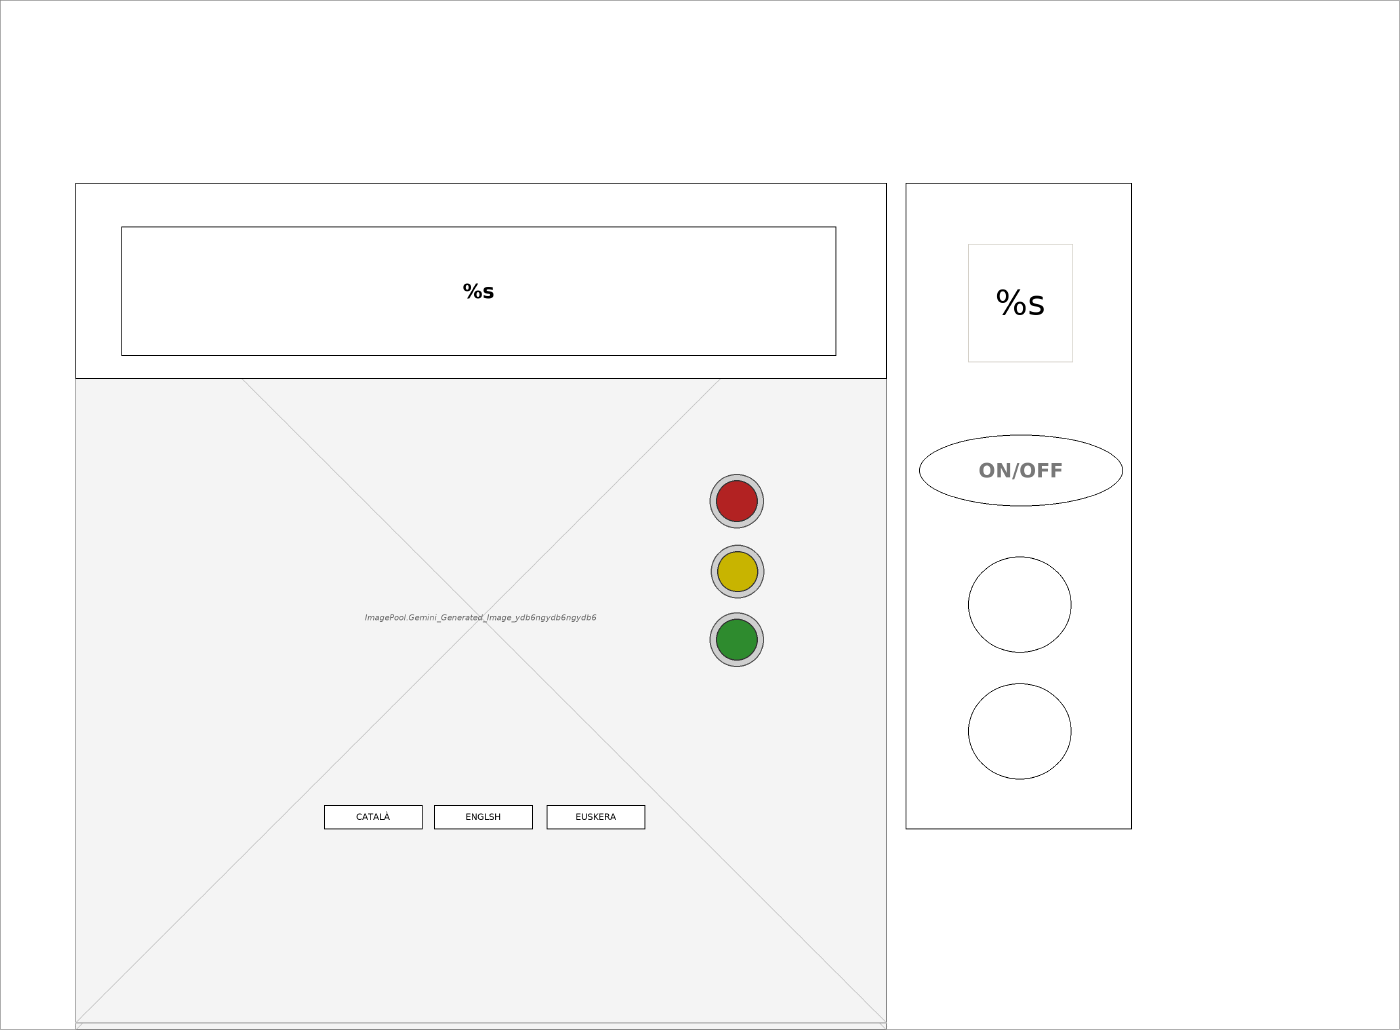
VISUALIZATION mainPage  // 1767x1301
    Image (95,272 1024x1024), invisible if: MAIN.boolENG, image: ImagePool.1772114357870
    RoundedRectangle (951,388 816x285), angle 90
    Image (95,253 1024x1048), invisible if: MAIN.boolCAT, image: ImagePool.Gemini_Generated_Image_6byr8p6byr8p6byr - copia
    Image (95,268 1024x1024), invisible if: MAIN.boolEUS, image: ImagePool.Gemini_Generated_Image_ydb6ngydb6ngydb6
    RoundedRectangle (95,231 1024x247)
    Lamp1 (890,593 80x80), variable: MAIN.mytrafficlight.outputs.REDlight, style: Lamp-Lamp1-Red
    Lamp1 (891,683 80x78), variable: MAIN.mytrafficlight.outputs.YELLOWlight, style: Lamp-Lamp1-Yellow
    Lamp1 (890,768 80x80), variable: MAIN.mytrafficlight.outputs.GREENlight, style: Lamp-Lamp1-Green
    Label (424,246 395x30), "EL HMI DEL SEMÁFORO"
    Ellipse (1222,703 130x121), colour toggle: MAIN.mytrafficlight.inputs.iGreen
        tap MAIN.mytrafficlight.inputs.iGreen
    Ellipse (1222,863 130x121), colour toggle: MAIN.mytrafficlight.inputs.iRed
        tap MAIN.mytrafficlight.inputs.iRed p1329445385=TRUE
    Ellipse (1160,549 257x90), "ON/OFF"
        toggle MAIN.updateState.HMI_Switch
    RoundedRectangle (409,1017 124x30), "CATALÀ"
        toggle MAIN.boolCAT
        OnMouseClick: ChangeLanguage ChangeLanguage=CATALÀ
        OnMouseClick: execute {
            MAIN.boolCAT := FALSE;
            MAIN.boolENG := TRUE;
            MAIN.boolEUS := TRUE;
        }
    RoundedRectangle (548,1017 124x30), "ENGLSH"
        OnMouseClick: ChangeLanguage ChangeLanguage=ENGLISH
        OnMouseClick: execute {
            MAIN.boolCAT := TRUE;
            MAIN.boolEUS := TRUE;
            MAIN.boolENG := FALSE;
        }
    RoundedRectangle (690,1017 124x30), "EUSKERA"
        toggle MAIN.boolEUS
        OnMouseClick: ChangeLanguage ChangeLanguage=EUSKERA
        OnMouseClick: execute {
            MAIN.boolCAT := TRUE;
            MAIN.boolENG := TRUE;
            MAIN.boolEUS := FALSE;
        }
    Textfield (1222,308 132x149), "%s", text variable: MAIN.visuTIME
        p4168582468: MAIN.visuTIME
    Rectangle (153,286 902x163), "%s", text list: 'GlobalTextList', text index: MAIN.mensajeIdioma
END_VISUALIZATION

(* stored: Version 1.1.0.1
   Visu mainPage: Id {438d3a89-436e-454b-9d50-699fc3e0c00f} *)
